KUKA KRL program: P01pick1_2_antes.src, P01pick1_2_antes.dat

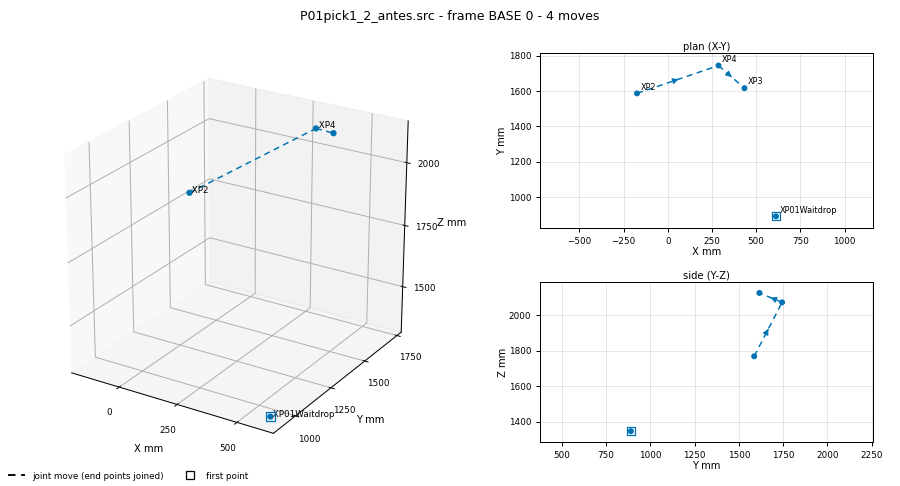
[picture p0: tool path of P01pick1_2_antes.src in frame BASE 0, 4 of 7 moves have a stored position in this frame; points joined in program order, loops and branches not executed]
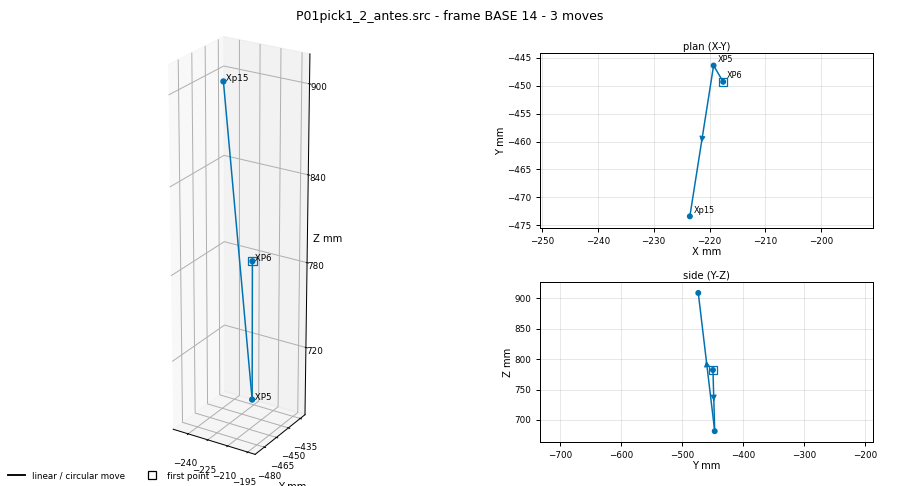
[picture p1: tool path of P01pick1_2_antes.src in frame BASE 14, 3 of 7 moves have a stored position in this frame; points joined in program order, loops and branches not executed]
--- P01pick1_2_antes.src ---
&ACCESS RVO1
&COMMENT Pick CARTON
&PARAM EDITMASK = *
&PARAM TEMPLATE = C:\KRC\Roboter\Template\vorgabe
&PARAM DISKPATH = KRC:\R1\Program\Sub Programs
DEF P01pick1_2_antes( )
;FOLD INI
  ;FOLD BASISTECH INI
BACKJUMP=FALSE
    GLOBAL INTERRUPT DECL 3 WHEN $STOPMESS==TRUE DO IR_STOPM ( )
    INTERRUPT ON 3
    BAS (#INITMOV,0 )
  ;ENDFOLD (BASISTECH INI)
;ENDFOLD (INI)
;================================================
; MODEL    : XXXX
; IE GROUP : XX
; STATION  : XXX
; ROBOT    : RX
; FUNCTION : pick Part in StXX
;================================================

;wait point

;FOLD PTP P01Waitdrop CONT Vel=100 % PDAT1 Tool[5] Base[0];%{PE}%R 8.3.48,%MKUKATPBASIS,%CMOVE,%VPTP,%P 1:PTP, 2:P01Waitdrop, 3:C_DIS, 5:100, 7:PDAT1
$BWDSTART=FALSE
PDAT_ACT=PPDAT1
FDAT_ACT=FP01Waitdrop
BAS(#PTP_PARAMS,100)
PTP XP01Waitdrop C_DIS
;ENDFOLD

;FOLD SYN OUT 241 'cil ventosas reposo' State=FALSE at START Delay=0 ms;%{PE}%R 8.3.48,%MKUKATPBASIS,%COUT,%VSYNOUT,%P 2:241, 3:cil ventosas reposo, 5:FALSE, 7:0, 9:0, 12:0
TRIGGER WHEN DISTANCE=0 DELAY=0 DO $OUT[241]=FALSE
;ENDFOLD
;FOLD SYN OUT 242 'cil ventosas activo' State=TRUE at START Delay=0 ms;%{PE}%R 8.3.48,%MKUKATPBASIS,%COUT,%VSYNOUT,%P 2:242, 3:cil ventosas activo, 5:TRUE, 7:0, 9:0, 12:0
TRIGGER WHEN DISTANCE=0 DELAY=0 DO $OUT[242]=TRUE
;ENDFOLD
;FOLD Fordtech.Tool_Req Tool Request: 2 ;%{PE}%MKUKATPUSER

Tool_Req (2)

;ENDFOLD
;FOLD Fordtech.Wait_Tool_Ready Wait Tool Ready: 2 ;%{PE}%MKUKATPUSER

Wait_Tool_Ready (2)

;ENDFOLD
;Wait For Area / Goto Safety / Return To Home


;FOLD ALTUA BASE
level1=PISO
BASE_DATA[11].Z=(ALTURA1*LEVEL1)
BASE_DATA[14].Z=(ALTURA1*LEVEL1)

;ENDFOLD

;FOLD PTP P6 CONT Vel=100 % PDAT8 Tool[5] Base[14];%{PE}%R 8.3.48,%MKUKATPBASIS,%CMOVE,%VPTP,%P 1:PTP, 2:P6, 3:C_DIS, 5:100, 7:PDAT8
$BWDSTART=FALSE
PDAT_ACT=PPDAT8
FDAT_ACT=FP6
BAS(#PTP_PARAMS,100)
PTP XP6 C_DIS
;ENDFOLD
CONTINUE
CIL_VENT_ACTIVO()

;FOLD TORQMON SetLimits Axis1: 15 % Axis2: 20 % Axis3: 15 % Axis4: 15 % Axis5: 15 % Axis6: 15 %;%{PE}%R 8.3.48,%MKUKATPBASIS,%CTQ_MON,%VTQ_LIMITS,%P 2:TQ_LIMITS, 4:15, 7:20, 10:15, 13:15, 16:15, 19:15
SET_TQ_VALUES (15,20,15,15,15,15)
;ENDFOLD

;FOLD LIN P5 Vel=0.5 m/s CPDAT6 Tool[5] Base[14];%{PE}%R 8.3.48,%MKUKATPBASIS,%CMOVE,%VLIN,%P 1:LIN, 2:P5, 3:, 5:0.5, 7:CPDAT6
$BWDSTART=FALSE
LDAT_ACT=LCPDAT6
FDAT_ACT=FP5
BAS(#CP_PARAMS,0.5)
LIN XP5
;ENDFOLD
SUCTION_ON()

;FOLD WAIT Time=2 sec;%{PE}%R 8.3.48,%MKUKATPBASIS,%CWAIT,%VWAIT,%P 3:2
WAIT SEC 2
;ENDFOLD

;FOLD LIN p15 CONT Vel=0.15 m/s L Tool[5] Base[14];%{PE}%R 8.3.48,%MKUKATPBASIS,%CMOVE,%VLIN,%P 1:LIN, 2:p15, 3:C_DIS C_DIS, 5:0.15, 7:L
$BWDSTART=FALSE
LDAT_ACT=LL
FDAT_ACT=Fp15
BAS(#CP_PARAMS,0.15)
LIN Xp15 C_DIS C_DIS
;ENDFOLD

;FOLD WAIT FOR ( IN 60 'Vacum ok' ) CONT;%{PE}%R 8.3.48,%MKUKATPBASIS,%CEXT_WAIT_FOR,%VEXT_WAIT_FOR,%P 2:, 4:, 5:$IN, 6:60, 7:Vacum ok, 9:CONTINUE
CONTINUE
WAIT FOR  ( $IN[60] )
;ENDFOLD

;FOLD PTP P2 CONT Vel=50 % L Tool[5] Base[0];%{PE}%R 8.3.48,%MKUKATPBASIS,%CMOVE,%VPTP,%P 1:PTP, 2:P2, 3:C_DIS, 5:50, 7:L
$BWDSTART=FALSE
PDAT_ACT=PL
FDAT_ACT=FP2
BAS(#PTP_PARAMS,50)
PTP XP2 C_DIS
;ENDFOLD

;FOLD Fordtech.Job_Rdy Set Job Ready: 5 ;%{PE}%MKUKATPUSER

Job_Ready (5)

;ENDFOLD

;Deja torqmon a valores nominales
SET_TQ_VALUES ( )

;FOLD PTP P4 CONT Vel=50 % L Tool[0] Base[0];%{PE}%R 8.3.48,%MKUKATPBASIS,%CMOVE,%VPTP,%P 1:PTP, 2:P4, 3:C_DIS, 5:50, 7:L
$BWDSTART=FALSE
PDAT_ACT=PL
FDAT_ACT=FP4
BAS(#PTP_PARAMS,50)
PTP XP4 C_DIS
;ENDFOLD


;FOLD SYN OUT 17 'Area Release 1' State=TRUE at START Delay=0 ms;%{PE}%R 8.3.48,%MKUKATPBASIS,%COUT,%VSYNOUT,%P 2:17, 3:Area Release 1, 5:TRUE, 7:0, 9:0, 12:0
TRIGGER WHEN DISTANCE=0 DELAY=0 DO $OUT[17]=TRUE
;ENDFOLD

;FOLD PTP P3 CONT Vel=100 % PDAT6 Tool[0] Base[0];%{PE}%R 8.3.48,%MKUKATPBASIS,%CMOVE,%VPTP,%P 1:PTP, 2:P3, 3:C_DIS, 5:100, 7:PDAT6
$BWDSTART=FALSE
PDAT_ACT=PPDAT6
FDAT_ACT=FP3
BAS(#PTP_PARAMS,100)
PTP XP3 C_DIS
;ENDFOLD

;FOLD TYPE INFO

O_TYPE_REQ=FALSE
WAIT FOR I_TYPE_INFO==0
O_TYPE_REQ=TRUE
WAIT FOR (I_TYPE_INFO>0)
O_TYPE_INFO=I_TYPE_INFO
POS_CARTON=I_TYPE_INFO
O_TYPE_REQ=FALSE


;ENDFOLD


;FOLD WAIT FOR ( IN 20 'Area 4 Ready' );%{PE}%R 8.3.48,%MKUKATPBASIS,%CEXT_WAIT_FOR,%VEXT_WAIT_FOR,%P 2:, 4:, 5:$IN, 6:20, 7:Area 4 Ready, 9:
WAIT FOR  ( $IN[20] )
;ENDFOLD
;FOLD OUT 20 'Area Release 4' State=FALSE ;%{PE}%R 8.3.48,%MKUKATPBASIS,%COUT,%VOUTX,%P 2:20, 3:Area Release 4, 5:FALSE, 6:
$OUT[20]=FALSE
;ENDFOLD

;Jump Adress
PEXIT:


END

--- P01pick1_2_antes.dat ---
&ACCESS RVO1
&COMMENT Pick CARTON
&PARAM EDITMASK = *
&PARAM TEMPLATE = C:\KRC\Roboter\Template\vorgabe
&PARAM DISKPATH = KRC:\R1\Program\Sub Programs
DEFDAT P01pick1_2_antes

EXT  BAS (BAS_COMMAND  :IN,REAL  :IN )
DECL INT SUCCESS
;******************************
;*     E6POS Declarations     *
;******************************

DECL E6POS XP01WAITREQ2={X 2157.35596,Y -301.755188,Z 2852.14893,A -15.8183,B 72.8074417,C -9.82211304,S 2,T 34,E1 0.0,E2 0.0,E3 0.0,E4 0.0,E5 0.0,E6 0.0}
DECL E6POS XP10={X 2411.43896,Y 1748.73096,Z -1095.62903,A -177.692307,B -16.9195194,C 42.7874298,S 2,T 34,E1 0.0,E2 0.0,E3 0.0,E4 0.0,E5 0.0,E6 0.0}
DECL E6POS XP20={X 1670.59900,Y -157.831207,Z 2354.64209,A -15.8183,B 72.8074417,C -9.82211304,S 2,T 34,E1 0.0,E2 0.0,E3 0.0,E4 0.0,E5 0.0,E6 0.0}
DECL E6POS XP30={X 1670.59900,Y -157.831207,Z 2354.64209,A -15.8183,B 72.8074417,C -9.82211304,S 2,T 34,E1 0.0,E2 0.0,E3 0.0,E4 0.0,E5 0.0,E6 0.0}
DECL E6POS XDROP_POS={X 1670.59900,Y -157.831207,Z 2354.64209,A -15.8183,B 72.8074417,C -9.82211304,S 2,T 34,E1 0.0,E2 0.0,E3 0.0,E4 0.0,E5 0.0,E6 0.0}
DECL E6POS XP40={X 2411.43896,Y 1748.73096,Z -1095.62903,A -177.692307,B -16.9195194,C 42.7874298,S 2,T 34,E1 0.0,E2 0.0,E3 0.0,E4 0.0,E5 0.0,E6 0.0}
DECL E6POS XP50={X 2411.43896,Y 1748.73096,Z -1095.62903,A -177.692307,B -16.9195194,C 42.7874298,S 2,T 34,E1 0.0,E2 0.0,E3 0.0,E4 0.0,E5 0.0,E6 0.0}
DECL E6POS XP01WAITREL2={X 2411.43896,Y 1748.73096,Z -1095.62903,A -177.692307,B -16.9195194,C 42.7874298,S 2,T 34,E1 0.0,E2 0.0,E3 0.0,E4 0.0,E5 0.0,E6 0.0}

;******************************
;*     FDAT Declarations      *
;******************************

DECL FDAT FP01WAITREQ2={TOOL_NO 12,BASE_NO 0,IPO_FRAME #BASE}
DECL FDAT FP10={TOOL_NO 12,BASE_NO 0,IPO_FRAME #TCP}
DECL FDAT FP20={TOOL_NO 12,BASE_NO 0,IPO_FRAME #TCP}
DECL FDAT FP30={TOOL_NO 12,BASE_NO 0,IPO_FRAME #TCP}
DECL FDAT FDROP_POS={TOOL_NO 12,BASE_NO 0,IPO_FRAME #TCP}
DECL FDAT FP40={TOOL_NO 12,BASE_NO 0,IPO_FRAME #TCP}
DECL FDAT FP50={TOOL_NO 12,BASE_NO 0,IPO_FRAME #TCP}
DECL FDAT FP01WAITREL2={TOOL_NO 12,BASE_NO 0,IPO_FRAME #TCP}

;******************************
;*  PDAT & LDAT Declarations  *
;******************************

DECL PDAT PH={VEL 100.000,ACC 100.000,APO_DIST 100.000,APO_MODE #CDIS,GEAR_JERK 100.000,EXAX_IGN 0}

DECL MODULEPARAM_T LAST_TP_PARAMS={PARAMS[] "FORDTECH.P_AREA_REQ=1; FORDTECH.P_SAFETY_POS=0; FORDTECH.P_RET=0; Kuka.VelocityFieldEnabled=True; Kuka.ColDetectFieldEnabled=True; Kuka.MovementParameterFieldEnabled=True; Kuka.IsAngleEnabled=False; Kuka.PointName=BATPOS13; Kuka.FrameData.base_no=0; Kuka.FrameData.tool_no=5; Kuka.FrameData.ipo_frame=#BASE; Kuka.isglobalpoint=False; Kuka.MoveDataPtpName=H; Kuka.MovementDataPdat.apo_mode=#CDIS; Kuka.MovementDataPdat.apo_dist=100; Kuka.MovementData.vel=100; Kuka.MovementData.acc=100; Kuka.MovementData.exax_ign=0; Kuka.VelocityPtp=100; Kuka.BlendingEnabled=False; Kuka.APXEnabled=False; Kuka.CurrentCDSetIndex=0; Kuka.FrameData.point2=; Kuka.MoveDataName=CPDAT2; Kuka.MovementData.cb={AUX_PT {ORI #CONSIDER,E1 #CONSIDER,E2 #CONSIDER,E3 #CONSIDER,E4 #CONSIDER,E5 #CONSIDER,E6 #CONSIDER},TARGET_PT {ORI #INTERPOLATE,E1 #INTERPOLATE,E2 #INTERPOLATE,E3 #INTERPOLATE,E4 #INTERPOLATE,E5 #INTERPOLATE,E6 #INTERPOLATE}}; Kuka.MovementData.apo_fac=50; Kuka.MovementData.apo_dist=500; Kuka.MovementData.axis_acc=100; Kuka.MovementData.axis_vel=100; Kuka.MovementData.circ_typ=#BASE; Kuka.MovementData.jerk_fac=50; Kuka.MovementData.ori_typ=#VAR; Kuka.VelocityPath=2  "}
DECL E6POS XP01Waitdrop={X 611.925903,Y 891.248230,Z 1346.61865,A -112.895660,B 8.25603676,C -175.944733,S 6,T 27,E1 0.0,E2 0.0,E3 0.0,E4 0.0,E5 0.0,E6 0.0}
DECL FDAT FP01Waitdrop={TOOL_NO 5,BASE_NO 0,IPO_FRAME #BASE,POINT2[] " ",TQ_STATE FALSE}
DECL E6POS XBATPOS1={X 290.951233,Y 816.177124,Z 1155.55042,A -86.9976196,B 22.0779018,C -179.006119,S 6,T 27,E1 0.0,E2 0.0,E3 0.0,E4 0.0,E5 0.0,E6 0.0}
DECL FDAT FBATPOS1={TOOL_NO 5,BASE_NO 11,IPO_FRAME #BASE,POINT2[] " "}
DECL E6POS XBATPOS2={X 763.140686,Y 824.200684,Z 1155.55042,A -86.9976196,B 22.0779018,C -179.006119,S 6,T 27,E1 0.0,E2 0.0,E3 0.0,E4 0.0,E5 0.0,E6 0.0}
DECL FDAT FBATPOS2={TOOL_NO 5,BASE_NO 11,IPO_FRAME #BASE,POINT2[] " "}
DECL E6POS XBATPOS3={X 290.951263,Y 1017.51129,Z 1155.55042,A -86.9976196,B 22.0779018,C -179.006119,S 6,T 27,E1 0.0,E2 0.0,E3 0.0,E4 0.0,E5 0.0,E6 0.0}
DECL FDAT FBATPOS3={TOOL_NO 5,BASE_NO 11,IPO_FRAME #BASE,POINT2[] " "}
DECL E6POS XBATPOS4={X 768.407043,Y 1017.51129,Z 1155.55042,A -86.9976196,B 22.0779018,C -179.006119,S 6,T 27,E1 0.0,E2 0.0,E3 0.0,E4 0.0,E5 0.0,E6 0.0}
DECL FDAT FBATPOS4={TOOL_NO 5,BASE_NO 11,IPO_FRAME #BASE,POINT2[] " "}
DECL E6POS XBATPOS5={X 290.951263,Y 1218.65857,Z 1155.55042,A -86.9976196,B 22.0779018,C -179.006119,S 6,T 27,E1 0.0,E2 0.0,E3 0.0,E4 0.0,E5 0.0,E6 0.0}
DECL FDAT FBATPOS5={TOOL_NO 5,BASE_NO 11,IPO_FRAME #BASE,POINT2[] " "}
DECL E6POS XBATPOS6={X 738.674316,Y 1202.54663,Z 1155.55042,A -86.9976196,B 22.0779018,C -179.006119,S 6,T 27,E1 0.0,E2 0.0,E3 0.0,E4 0.0,E5 0.0,E6 0.0}
DECL FDAT FBATPOS6={TOOL_NO 5,BASE_NO 11,IPO_FRAME #BASE,POINT2[] " "}
DECL E6POS XBATPOS7={X 290.951263,Y 1386.78320,Z 1155.55042,A -86.9976196,B 22.0779018,C -179.006119,S 6,T 27,E1 0.0,E2 0.0,E3 0.0,E4 0.0,E5 0.0,E6 0.0}
DECL FDAT FBATPOS7={TOOL_NO 5,BASE_NO 11,IPO_FRAME #BASE,POINT2[] " "}
DECL E6POS XBATPOS8={X 728.249,Y 1368.06873,Z 1155.55042,A -86.9976196,B 22.0779018,C -179.006119,S 6,T 27,E1 0.0,E2 0.0,E3 0.0,E4 0.0,E5 0.0,E6 0.0}
DECL FDAT FBATPOS8={TOOL_NO 5,BASE_NO 11,IPO_FRAME #BASE,POINT2[] " "}
DECL E6POS XBATPOS9={X 290.951263,Y 1572.31165,Z 1155.55042,A -86.9976196,B 22.0779018,C -179.006119,S 6,T 27,E1 0.0,E2 0.0,E3 0.0,E4 0.0,E5 0.0,E6 0.0}
DECL FDAT FBATPOS9={TOOL_NO 5,BASE_NO 11,IPO_FRAME #BASE,POINT2[] " "}
DECL E6POS XBATPOS10={X 753.970337,Y 1583.41736,Z 1155.55042,A -86.9976196,B 22.0779018,C -179.006119,S 6,T 27,E1 0.0,E2 0.0,E3 0.0,E4 0.0,E5 0.0,E6 0.0}
DECL FDAT FBATPOS10={TOOL_NO 5,BASE_NO 11,IPO_FRAME #BASE,POINT2[] " "}
DECL E6POS XBATPOS11={X 301.951050,Y 1774.17639,Z 1155.55042,A -86.9976196,B 22.0779018,C -179.006119,S 6,T 27,E1 0.0,E2 0.0,E3 0.0,E4 0.0,E5 0.0,E6 0.0}
DECL FDAT FBATPOS11={TOOL_NO 5,BASE_NO 11,IPO_FRAME #BASE,POINT2[] " "}
DECL E6POS XBATPOS12={X 738.848694,Y 1774.17639,Z 1155.55042,A -86.9976196,B 22.0779018,C -179.006119,S 6,T 27,E1 0.0,E2 0.0,E3 0.0,E4 0.0,E5 0.0,E6 0.0}
DECL FDAT FBATPOS12={TOOL_NO 5,BASE_NO 11,IPO_FRAME #BASE,POINT2[] " "}
DECL E6POS XBATPOS13={X -1007.42786,Y 1689.02979,Z 871.879700,A -90.0765839,B 0.159503683,C -179.722214,S 6,T 27,E1 0.0,E2 0.0,E3 0.0,E4 0.0,E5 0.0,E6 0.0}
DECL FDAT FBATPOS13={TOOL_NO 5,BASE_NO 0,IPO_FRAME #BASE,POINT2[] " "}
DECL LDAT LCPDAT1={VEL 2.00000,ACC 100.000,APO_DIST 500.000,APO_FAC 50.0000,AXIS_VEL 100.000,AXIS_ACC 100.000,ORI_TYP #VAR,CIRC_TYP #BASE,JERK_FAC 50.0000,GEAR_JERK 100.000,EXAX_IGN 0,CB {AUX_PT {ORI #CONSIDER,E1 #CONSIDER,E2 #CONSIDER,E3 #CONSIDER,E4 #CONSIDER,E5 #CONSIDER,E6 #CONSIDER},TARGET_PT {ORI #INTERPOLATE,E1 #INTERPOLATE,E2 #INTERPOLATE,E3 #INTERPOLATE,E4 #INTERPOLATE,E5 #INTERPOLATE,E6 #INTERPOLATE}}}
DECL E6POS XBATPOS14={X -1007.42786,Y 1689.02979,Z 763.563721,A -90.0765839,B 0.159503683,C -179.722214,S 6,T 27,E1 0.0,E2 0.0,E3 0.0,E4 0.0,E5 0.0,E6 0.0}
DECL FDAT FBATPOS14={TOOL_NO 5,BASE_NO 0,IPO_FRAME #BASE,POINT2[] " "}
DECL LDAT LCPDAT2={VEL 2.00000,ACC 100.000,APO_DIST 500.000,APO_FAC 50.0000,AXIS_VEL 100.000,AXIS_ACC 100.000,ORI_TYP #VAR,CIRC_TYP #BASE,JERK_FAC 50.0000,GEAR_JERK 100.000,EXAX_IGN 0,CB {AUX_PT {ORI #CONSIDER,E1 #CONSIDER,E2 #CONSIDER,E3 #CONSIDER,E4 #CONSIDER,E5 #CONSIDER,E6 #CONSIDER},TARGET_PT {ORI #INTERPOLATE,E1 #INTERPOLATE,E2 #INTERPOLATE,E3 #INTERPOLATE,E4 #INTERPOLATE,E5 #INTERPOLATE,E6 #INTERPOLATE}}}
DECL BASIS_SUGG_T LAST_BASIS={POINT1[] "P0                      ",POINT2[] "P0                      ",CP_PARAMS[] "CPDAT0                  ",PTP_PARAMS[] "PDAT0                   ",CONT[] "                        ",CP_VEL[] "0.15                    ",PTP_VEL[] "100                     ",SYNC_PARAMS[] "SYNCDAT                 ",SPL_NAME[] "S0                      ",A_PARAMS[] "ADAT0                   "}
DECL E6POS XP01WAIRDROP={X -1019.53113,Y 1662.02271,Z 1494.18042,A -87.0150,B 22.0766449,C -179.006226,S 6,T 27,E1 0.0,E2 0.0,E3 0.0,E4 0.0,E5 0.0,E6 0.0}
DECL FDAT FP01Wairdrop={TOOL_NO 12,BASE_NO 0,IPO_FRAME #BASE,POINT2[] " ",TQ_STATE FALSE}
DECL PDAT PPDAT1={VEL 100.000,ACC 100.000,APO_DIST 100.000,APO_MODE #CDIS,GEAR_JERK 50.0000,EXAX_IGN 0}
DECL PDAT PPDAT2={VEL 100.000,ACC 100.000,APO_DIST 100.000,GEAR_JERK 50.0000,EXAX_IGN 0}
DECL LDAT LCPDAT3={VEL 2.00000,ACC 100.000,APO_DIST 100.000,APO_FAC 50.0000,AXIS_VEL 100.000,AXIS_ACC 100.000,ORI_TYP #VAR,CIRC_TYP #BASE,JERK_FAC 50.0000,GEAR_JERK 50.0000,EXAX_IGN 0}
DECL E6POS XWAITDROP={X -1019.53113,Y 1662.02271,Z 1494.18042,A -87.0150,B 22.0766449,C -179.006226,S 6,T 27,E1 0.0,E2 0.0,E3 0.0,E4 0.0,E5 0.0,E6 0.0}
DECL FDAT FWaitdrop={TOOL_NO 5,BASE_NO 0,IPO_FRAME #BASE,POINT2[] " ",TQ_STATE FALSE}
DECL PDAT PPDAT3={VEL 100.000,ACC 100.000,APO_DIST 100.000,GEAR_JERK 50.0000,EXAX_IGN 0}
DECL E6POS XP01={X -1224.93213,Y 1500.55322,Z 894.067444,A -88.3210297,B -0.0488793,C 179.376755,S 6,T 27,E1 0.0,E2 0.0,E3 0.0,E4 0.0,E5 0.0,E6 0.0}
DECL FDAT Fp01={TOOL_NO 5,BASE_NO 0,IPO_FRAME #BASE,POINT2[] " ",TQ_STATE FALSE}
DECL LDAT LCPDAT4={VEL 2.00000,ACC 100.000,APO_DIST 100.000,APO_FAC 50.0000,AXIS_VEL 100.000,AXIS_ACC 100.000,ORI_TYP #VAR,CIRC_TYP #BASE,JERK_FAC 50.0000,GEAR_JERK 50.0000,EXAX_IGN 0}
DECL E6POS XP02={X -1224.93213,Y 1500.55322,Z 1010.30774,A -88.3210297,B -0.0488792881,C 179.376755,S 6,T 27,E1 0.0,E2 0.0,E3 0.0,E4 0.0,E5 0.0,E6 0.0}
DECL FDAT Fp02={TOOL_NO 5,BASE_NO 0,IPO_FRAME #BASE,POINT2[] " ",TQ_STATE FALSE}
DECL PDAT PPDAT4={VEL 100.000,ACC 100.000,APO_DIST 100.000,APO_MODE #CDIS,GEAR_JERK 50.0000,EXAX_IGN 0}
DECL E6POS XP1={X -1287.24158,Y 1504.14661,Z 1245.59644,A -89.5973740,B -0.0771145225,C -179.659088,S 6,T 27,E1 0.0,E2 0.0,E3 0.0,E4 0.0,E5 0.0,E6 0.0}
DECL FDAT FP1={TOOL_NO 5,BASE_NO 0,IPO_FRAME #BASE,POINT2[] " ",TQ_STATE FALSE}
DECL LDAT LCPDAT5={VEL 2.00000,ACC 100.000,APO_DIST 100.000,APO_FAC 50.0000,AXIS_VEL 100.000,AXIS_ACC 100.000,ORI_TYP #VAR,CIRC_TYP #BASE,JERK_FAC 50.0000,GEAR_JERK 50.0000,EXAX_IGN 0}
DECL E6POS XP2={X -173.782318,Y 1586.64294,Z 1769.31897,A -80.7608490,B 1.54349911,C -104.851402,S 6,T 27,E1 0.0,E2 0.0,E3 0.0,E4 0.0,E5 0.0,E6 0.0}
DECL FDAT FP2={TOOL_NO 5,BASE_NO 0,IPO_FRAME #BASE,POINT2[] " ",TQ_STATE FALSE}
DECL PDAT PPDAT5={VEL 100.000,ACC 100.000,APO_DIST 100.000,APO_MODE #CDIS,GEAR_JERK 50.0000,EXAX_IGN 0}
DECL E6POS XP3={X 433.858368,Y 1615.89539,Z 2126.45166,A -90.5571899,B 1.60751188,C -89.4436417,S 6,T 27,E1 0.0,E2 0.0,E3 0.0,E4 0.0,E5 0.0,E6 0.0}
DECL FDAT FP3={TOOL_NO 0,BASE_NO 0,IPO_FRAME #BASE,POINT2[] " ",TQ_STATE FALSE}
DECL PDAT PPDAT6={VEL 100.000,ACC 100.000,APO_DIST 100.000,APO_MODE #CDIS,GEAR_JERK 50.0000,EXAX_IGN 0}
DECL E6POS XP4={X 286.791199,Y 1744.11914,Z 2073.52808,A -80.6430283,B -0.415123552,C -92.9314499,S 6,T 27,E1 0.0,E2 0.0,E3 0.0,E4 0.0,E5 0.0,E6 0.0}
DECL FDAT FP4={TOOL_NO 0,BASE_NO 0,IPO_FRAME #BASE,POINT2[] " ",TQ_STATE FALSE}
DECL PDAT PPDAT7={VEL 100.000,ACC 100.000,APO_DIST 100.000,APO_MODE #CDIS,GEAR_JERK 50.0000,EXAX_IGN 0}
DECL E6POS XP5={X -219.270447,Y -446.384949,Z 681.601868,A -90.5906143,B -0.937737823,C -179.576187,S 6,T 27,E1 0.0,E2 0.0,E3 0.0,E4 0.0,E5 0.0,E6 0.0}
DECL FDAT FP5={TOOL_NO 5,BASE_NO 14,IPO_FRAME #BASE,POINT2[] " ",TQ_STATE FALSE}
DECL LDAT LCPDAT6={VEL 2.00000,ACC 100.000,APO_DIST 100.000,APO_FAC 50.0000,AXIS_VEL 100.000,AXIS_ACC 100.000,ORI_TYP #VAR,CIRC_TYP #BASE,JERK_FAC 50.0000,GEAR_JERK 50.0000,EXAX_IGN 0}
DECL E6POS XP6={X -217.555786,Y -449.303436,Z 782.114868,A -91.2796783,B -1.08149838,C -179.690292,S 6,T 27,E1 0.0,E2 0.0,E3 0.0,E4 0.0,E5 0.0,E6 0.0}
DECL FDAT FP6={TOOL_NO 5,BASE_NO 14,IPO_FRAME #BASE,POINT2[] " ",TQ_STATE FALSE}
DECL PDAT PPDAT8={VEL 100.000,ACC 100.000,APO_DIST 100.000,APO_MODE #CDIS,GEAR_JERK 50.0000,EXAX_IGN 0}
DECL E6POS XP7={X -1287.24158,Y 1504.14661,Z 1245.59644,A -89.5973740,B -0.0771145225,C -179.659088,S 6,T 27,E1 0.0,E2 0.0,E3 0.0,E4 0.0,E5 0.0,E6 0.0}
DECL FDAT FP7={TOOL_NO 5,BASE_NO 0,IPO_FRAME #BASE,POINT2[] " ",TQ_STATE FALSE}
DECL LDAT LCPDAT7={VEL 2.00000,ACC 100.000,APO_DIST 100.000,APO_FAC 50.0000,AXIS_VEL 100.000,AXIS_ACC 100.000,ORI_TYP #VAR,CIRC_TYP #BASE,JERK_FAC 50.0000,GEAR_JERK 50.0000,EXAX_IGN 0}
DECL E6POS XP8={X -1287.24158,Y 1504.14661,Z 1245.59644,A -89.5973740,B -0.0771145225,C -179.659088,S 6,T 27,E1 0.0,E2 0.0,E3 0.0,E4 0.0,E5 0.0,E6 0.0}
DECL FDAT FP8={TOOL_NO 5,BASE_NO 0,IPO_FRAME #BASE,POINT2[] " ",TQ_STATE FALSE}
DECL LDAT LCPDAT8={VEL 2.00000,ACC 100.000,APO_DIST 100.000,APO_FAC 50.0000,AXIS_VEL 100.000,AXIS_ACC 100.000,ORI_TYP #VAR,CIRC_TYP #BASE,JERK_FAC 50.0000,GEAR_JERK 50.0000,EXAX_IGN 0}
DECL E6POS XP9={X -1287.24158,Y 1504.14661,Z 1245.59644,A -89.5973740,B -0.0771145225,C -179.659088,S 6,T 27,E1 0.0,E2 0.0,E3 0.0,E4 0.0,E5 0.0,E6 0.0}
DECL FDAT FP9={TOOL_NO 5,BASE_NO 0,IPO_FRAME #BASE,POINT2[] " ",TQ_STATE FALSE}
DECL LDAT LCPDAT9={VEL 2.00000,ACC 100.000,APO_DIST 100.000,APO_FAC 50.0000,AXIS_VEL 100.000,AXIS_ACC 100.000,ORI_TYP #VAR,CIRC_TYP #BASE,JERK_FAC 50.0000,GEAR_JERK 50.0000,EXAX_IGN 0}
DECL E6POS XP11={X -1287.24158,Y 1504.14661,Z 1245.59644,A -89.5973740,B -0.0771145225,C -179.659088,S 6,T 27,E1 0.0,E2 0.0,E3 0.0,E4 0.0,E5 0.0,E6 0.0}
DECL FDAT FP11={TOOL_NO 5,BASE_NO 0,IPO_FRAME #BASE,POINT2[] " ",TQ_STATE FALSE}
DECL LDAT LCPDAT10={VEL 2.00000,ACC 100.000,APO_DIST 100.000,APO_FAC 50.0000,AXIS_VEL 100.000,AXIS_ACC 100.000,ORI_TYP #VAR,CIRC_TYP #BASE,JERK_FAC 50.0000,GEAR_JERK 50.0000,EXAX_IGN 0}
DECL E6POS XP12={X -1287.24158,Y 1504.14661,Z 1245.59644,A -89.5973740,B -0.0771145225,C -179.659088,S 6,T 27,E1 0.0,E2 0.0,E3 0.0,E4 0.0,E5 0.0,E6 0.0}
DECL FDAT FP12={TOOL_NO 5,BASE_NO 0,IPO_FRAME #BASE,POINT2[] " ",TQ_STATE FALSE}
DECL LDAT LCPDAT11={VEL 2.00000,ACC 100.000,APO_DIST 100.000,APO_FAC 50.0000,AXIS_VEL 100.000,AXIS_ACC 100.000,ORI_TYP #VAR,CIRC_TYP #BASE,JERK_FAC 50.0000,GEAR_JERK 50.0000,EXAX_IGN 0}
DECL PDAT PPDAT0={VEL 100.000,ACC 100.000,APO_DIST 100.000,APO_MODE #CDIS,GEAR_JERK 50.0000,EXAX_IGN 0}
DECL E6POS XP0={X -1224.93213,Y 1500.55322,Z 890.307739,A -88.3210297,B -0.0488792881,C 179.376755,S 6,T 27,E1 0.0,E2 0.0,E3 0.0,E4 0.0,E5 0.0,E6 0.0}
DECL FDAT FP0={TOOL_NO 5,BASE_NO 11,IPO_FRAME #BASE,POINT2[] " ",TQ_STATE FALSE}
DECL E6POS Xp15={X -223.523224,Y -473.393524,Z 908.652832,A -90.6026688,B -1.36748445,C 179.369080,S 6,T 27,E1 0.0,E2 0.0,E3 0.0,E4 0.0,E5 0.0,E6 0.0}
DECL FDAT Fp15={TOOL_NO 5,BASE_NO 14,IPO_FRAME #BASE,POINT2[] " ",TQ_STATE FALSE}
DECL LDAT LCPDAT12={VEL 2.00000,ACC 100.000,APO_DIST 100.000,APO_FAC 50.0000,AXIS_VEL 100.000,AXIS_ACC 100.000,ORI_TYP #VAR,CIRC_TYP #BASE,JERK_FAC 50.0000,GEAR_JERK 50.0000,EXAX_IGN 0}
DECL LDAT LL={VEL 2.00000,ACC 25.0000,APO_DIST 100.000,APO_FAC 50.0000,AXIS_VEL 100.000,AXIS_ACC 100.000,ORI_TYP #VAR,CIRC_TYP #BASE,JERK_FAC 50.0000,GEAR_JERK 50.0000,EXAX_IGN 0}
DECL PDAT PL={VEL 100.000,ACC 25.0000,APO_DIST 100.000,APO_MODE #CDIS,GEAR_JERK 50.0000,EXAX_IGN 0}
ENDDAT
